TYPE U_UMC_Lenze_Control :
UNION
	Output		: UINT;
	Data		: T_UMC_Lenze_Control;
END_UNION
END_TYPE

(* stored: Version 1.1.0.1, ProductVersion 3.1.0.19
   DUT U_UMC_Lenze_Control: Id {ee731394-96a1-4716-a04f-7fd149420a24} *)
